// TIA Portal V19 export
TYPE "LEXCHANGETRAY_typeConstraintWorkstationEm_interface"
// stored: Access Published
   STRUCT
      deliver : "LEXCHANGETRAY_typeConstraintWorkstation_deliver_interface";
      recieve : "LEXCHANGETRAY_typeConstraintWorkstationEm_recieve_interface";
   END_STRUCT;
END_TYPE
